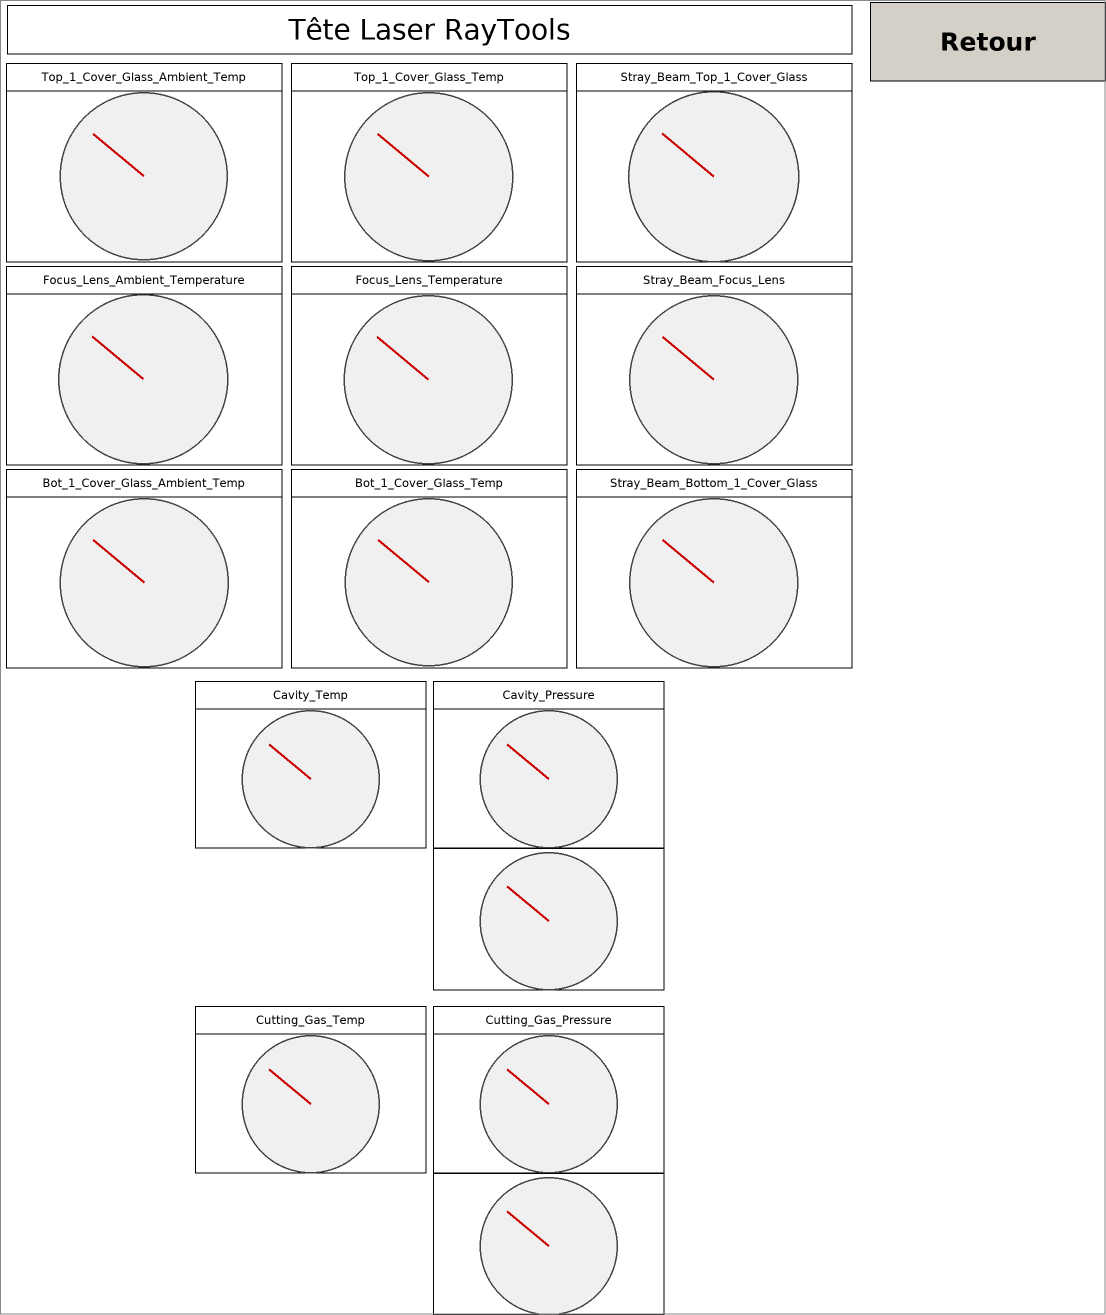
VISUALIZATION Laser_Tete_Raytools_2  // 1106x1315
    Rectangle (576,469 276x199)
    Rectangle (576,266 276x199)
    Rectangle (576,63 276x199)
    Rectangle (291,469 276x199)
    Rectangle (291,266 276x199)
    Rectangle (291,63 276x199)
    Rectangle (6,63 276x199)
    Rectangle (6,266 276x199)
    Rectangle (6,469 276x199)
    Meter (6,294 274x170), value: Data03_Focus_Lens_Ambient_Temperature/100, scale format: %.1f, scale 0..30
        p518627256: °C
    Rectangle (6,266 276x28), "Focus_Lens_Ambient_Temperature"
    Meter (291,295 274x169), value: Data04_Focus_Lens_Temperature/100, scale format: %.1f, scale 0..60
        p518627256: °C
    Rectangle (291,266 276x28), "Focus_Lens_Temperature"
    Meter (6,92 275x168), value: Data07_Top_1_Cover_Glass_Ambient_Temp/100, scale format: %.1f, scale 0..30
        p518627256: °C
    Rectangle (6,63 276x28), "Top_1_Cover_Glass_Ambient_Temp"
    Meter (292,92 273x169), value: Data08_Top_1_Cover_Glass_Temp/100, scale format: %.1f, scale 0..60
        p518627256: °C
    Rectangle (291,63 276x28), "Top_1_Cover_Glass_Temp"
    Meter (7,498 274x169), value: Data09_Bottom_1_Cover_Glass_Ambient_Temp/100, scale format: %.1f, scale 0..30
        p518627256: °C
    Rectangle (6,469 276x28), "Bot_1_Cover_Glass_Ambient_Temp"
    Meter (292,498 273x168), value: Data10_Bottom_1_Cover_Glasst_Temp/100, scale format: %.1f, scale 0..60
        p518627256: °C
    Rectangle (291,469 276x28), "Bot_1_Cover_Glass_Temp"
    Rectangle (195,681 231x167)
    Meter (195,710 231x138), value: Data11_Cavity_Temp/100, scale format: %.1f, scale 0..60
        p518627256: °C
    Rectangle (195,681 231x28), "Cavity_Temp"
    Rectangle (195,1006 231x167)
    Meter (195,1035 231x138), value: Data13_Cutting_Gas_Temp/100, scale format: %.1f, scale 0..60
        p518627256: °C
    Rectangle (195,1006 231x28), "Cutting_Gas_Temp"
    Rectangle (433,681 231x167)
    Meter (433,710 231x138), value: Data12_Cavity_Pressure/10, scale format: %.1f, scale 0..10
        p518627256: Bars
    Rectangle (433,681 231x28), "Cavity_Pressure"
    Rectangle (433,848 231x142)
    Meter (433,852 231x138), value: Data12_Cavity_Pressure/10, scale format: %.1f, scale 0..1
        p518627256: Bars
    Rectangle (433,1006 231x167)
    Meter (433,1035 231x138), value: Data14_Cutting_Gas_Pressure/10, scale format: %.1f, scale 0..10
        p518627256: Bars
    Rectangle (433,1006 231x28), "Cutting_Gas_Pressure"
    Rectangle (433,1173 231x142)
    Meter (433,1177 231x138), value: Data14_Cutting_Gas_Pressure/10, scale format: %.1f, scale 0..1
        p518627256: Bars
    Meter (577,91 273x171), value: Data27_Stray_Beam_Top_1_Cover_Glass/100, scale format: %.1f, scale 0..30
        p518627256: °C
    Rectangle (576,63 276x28), "Stray_Beam_Top_1_Cover_Glass"
    Meter (577,295 273x169), value: Data28_Stray_Beam_Focus_Lens/100, scale format: %.1f, scale 0..30
        p518627256: °C
    Rectangle (576,266 276x28), "Stray_Beam_Focus_Lens"
    Meter (577,498 273x169), value: Data29_Stray_Beam_Bottom_1_Cover_Glass/100, scale format: %.1f, scale 0..30
        p518627256: °C
    Rectangle (576,469 276x28), "Stray_Beam_Bottom_1_Cover_Glass"
    Rectangle (7,5 845x49), "Tête Laser RayTools"
    Rectangle (870,2 236x79), "Retour"
        OnMouseClick: change screen: Selection_Rep
        OnMouseClick: execute { Forcage_Rep.Num_Rep_Selectionne_pr_Forcage:=0; }
END_VISUALIZATION

(* stored: Version 1.1.0.1
   Visu Laser_Tete_Raytools_2: Id {edf31696-bec1-42e9-ba56-bc0435e16006} *)
